// TIA Portal project "FactoryIO_Template_S7-1200_V16_V16" (V16)
// Vorlageprojekt für das Buch mit Zielsystem S7-1200

(* hardware
DEVICE "S7-1200-Station_1"  S7-1200 Station
   slot 0: "Baugruppenträger_0"  Rack  V1.0
   slot 1: "PLC_1"  CPU 1211C DC/DC/DC  6ES7 211-1AE40-0XB0  V4.1
*)

// ===== PLC "PLC_1"  CPU 1211C DC/DC/DC =====

VAR_GLOBAL   // PLC tag table "Standard-Variablentabelle"
   "Start" AT %I0.0 : Bool;
   "stop" AT %I0.1 : Bool;
   "Vsion_top" AT %I0.2 : Bool;
   "Vision_base" AT %I0.3 : Bool;
   "Pusher_front_L_base" AT %I0.4 : Bool;
   "Pusher_back_L_base" AT %I0.5 : Bool;
   "Pusher_front_L_top" AT %I0.6 : Bool;
   "Pusher_back_L_top" AT %I0.7 : Bool;
   "Diff_base_pusher" AT %I1.0 : Bool;
   "Diff_top_pusher" AT %I1.1 : Bool;
   "clamped_base" AT %I1.2 : Bool;
   "clamped_top" AT %I1.3 : Bool;
   "Diff_Item_arm" AT %I1.4 : Bool;
   "Move_Z_sensor" AT %I1.5 : Bool;
   "Move_X_sensor" AT %I1.6 : Bool;
   "Diff_base_clamp" AT %I1.7 : Bool;
   "Diff_top_clamp" AT %I2.0 : Bool;
   "Diff_item_leave" AT %I2.1 : Bool;
   "belte_main" AT %Q0.0 : Bool;
   "belte_pushers" AT %Q0.1 : Bool;
   "pusher_base" AT %Q0.2 : Bool;
   "Pusher_top" AT %Q0.3 : Bool;
   "Belte_base" AT %Q0.4 : Bool;
   "Belte_top" AT %Q0.5 : Bool;
   "clamp_base" AT %Q0.6 : Bool;
   "clamp_top" AT %Q0.7 : Bool;
   "up_base" AT %Q1.0 : Bool;
   "Move_z" AT %Q1.1 : Bool;
   "Move_x" AT %Q1.2 : Bool;
   "Grap" AT %Q1.3 : Bool;
   "X" AT %M0.0 : Bool;
   "base" AT %M0.1 : Bool;
   "top" AT %M0.2 : Bool;
   "leave" AT %M0.3 : Bool;
END_VAR

// folder: System blocks/Program resources

DATA_BLOCK "hold_base"   // DB1
{ S7_Optimized_Access := 'TRUE' }
AUTHOR : Simatic
FAMILY : IEC
NAME : IEC_TMR
VERSION : 1.0
// stored: InstanceOfName IEC_TIMER
"IEC_TIMER"
BEGIN
END_DATA_BLOCK

DATA_BLOCK "hold_top"   // DB2
{ S7_Optimized_Access := 'TRUE' }
AUTHOR : Simatic
FAMILY : IEC
NAME : IEC_TMR
VERSION : 1.0
// stored: InstanceOfName IEC_TIMER
"IEC_TIMER"
BEGIN
END_DATA_BLOCK

DATA_BLOCK "wait_for Grap"   // DB3
{ S7_Optimized_Access := 'TRUE' }
AUTHOR : Simatic
FAMILY : IEC
NAME : IEC_TMR
VERSION : 1.0
// stored: InstanceOfName IEC_TIMER
"IEC_TIMER"
BEGIN
END_DATA_BLOCK

DATA_BLOCK "hold_down"   // DB4
{ S7_Optimized_Access := 'TRUE' }
AUTHOR : Simatic
FAMILY : IEC
NAME : IEC_TMR
VERSION : 1.0
// stored: InstanceOfName IEC_TIMER
"IEC_TIMER"
BEGIN
END_DATA_BLOCK

DATA_BLOCK "hold_clamp"   // DB5
{ S7_Optimized_Access := 'TRUE' }
AUTHOR : Simatic
FAMILY : IEC
NAME : IEC_TMR
VERSION : 1.0
// stored: InstanceOfName IEC_TIMER
"IEC_TIMER"
BEGIN
END_DATA_BLOCK

DATA_BLOCK "hlod_base"   // DB6
{ S7_Optimized_Access := 'TRUE' }
AUTHOR : Simatic
FAMILY : IEC
NAME : IEC_TMR
VERSION : 1.0
// stored: InstanceOfName IEC_TIMER
"IEC_TIMER"
BEGIN
END_DATA_BLOCK

DATA_BLOCK "up_hold"   // DB7
{ S7_Optimized_Access := 'TRUE' }
AUTHOR : Simatic
FAMILY : IEC
NAME : IEC_TMR
VERSION : 1.0
// stored: InstanceOfName IEC_TIMER
"IEC_TIMER"
BEGIN
END_DATA_BLOCK

DATA_BLOCK "hold_leave"   // DB8
{ S7_Optimized_Access := 'TRUE' }
AUTHOR : Simatic
FAMILY : IEC
NAME : IEC_TMR
VERSION : 1.0
// stored: InstanceOfName IEC_TIMER
"IEC_TIMER"
BEGIN
END_DATA_BLOCK

// folder: (top level)

FUNCTION "MHJ-PLC-Lab-Function-S71200" : Void   // FC9000, SCL
{ S7_Optimized_Access := 'TRUE' }
VERSION : 0.1
   VAR_TEMP
      rdTimeReturn : Int;
      outputTime : DTL;
      SyncVal : Byte;
      forVal : Int;
      forVal_2 : Int;
      Value : Byte;
   END_VAR
   VAR CONSTANT
      CompVal : Byte := 16#34;
      Value_01 : Byte := 16#11;
      Value_01_DW : DWord := 16#A165_D992;
      Value_02_DW : DWord := 16#58BE_4401;
   END_VAR
BEGIN

   #Value:=PEEK(area := 16#82,
        dbNumber := 0,
        byteOffset := 511);
   #Value := #Value + 1;

   POKE(area := 16#82,
        dbNumber := 0,
        byteOffset := 511,
        value := #Value);

   POKE(area:=16#81,
        dbNumber:=0,
        byteOffset:=1016,
        value:=#Value_01_DW);
   POKE(area := 16#81,
        dbNumber := 0,
        byteOffset := 1020,
        value := #Value_02_DW);

   POKE(area := 16#81,
        dbNumber := 0,
        byteOffset := 511,
        value := B#16#00);

   FOR #forVal := 0 TO 120 DO
       FOR #forVal_2:=0 TO 10 DO
           #rdTimeReturn:=RD_SYS_T(#outputTime);
           #rdTimeReturn := WR_SYS_T(#outputTime);
           #rdTimeReturn := RD_SYS_T(#outputTime);
           #rdTimeReturn := WR_SYS_T(#outputTime);
       END_FOR;
       #SyncVal:= PEEK(area := 16#81,
                      dbNumber := 0,
                      byteOffset := 511);
       IF #SyncVal = #CompVal THEN
          GOTO M_1;
       END_IF;
   END_FOR;
   RETURN;

   M_1:
   POKE(area := 16#81,
        dbNumber := 0,
        byteOffset := 511,
        value := B#16#0);
END_FUNCTION

ORGANIZATION_BLOCK "Main"   // OB1, LAD, ProgramCycle
TITLE = "Main Program Sweep (Cycle)"
{ S7_Optimized_Access := 'TRUE' }
VERSION : 0.1
   VAR_INPUT
      Initial_Call : Bool;   // Initial call of this OB
      Remanence : Bool;   // =True, if remanent data are available
   END_VAR
   VAR_TEMP   // added for the SCL form of the ladder/FBD networks
      _w1 : Bool;
   END_VAR
BEGIN

REGION Network 1: Konnektierungsbaustein für PLC-Lab
   // Im Netzwerk 1 wird der Konnektierungsbaustein für PLC-Lab aufgerufen.
   // Dieser Aufruf darf nicht entfernt werden!
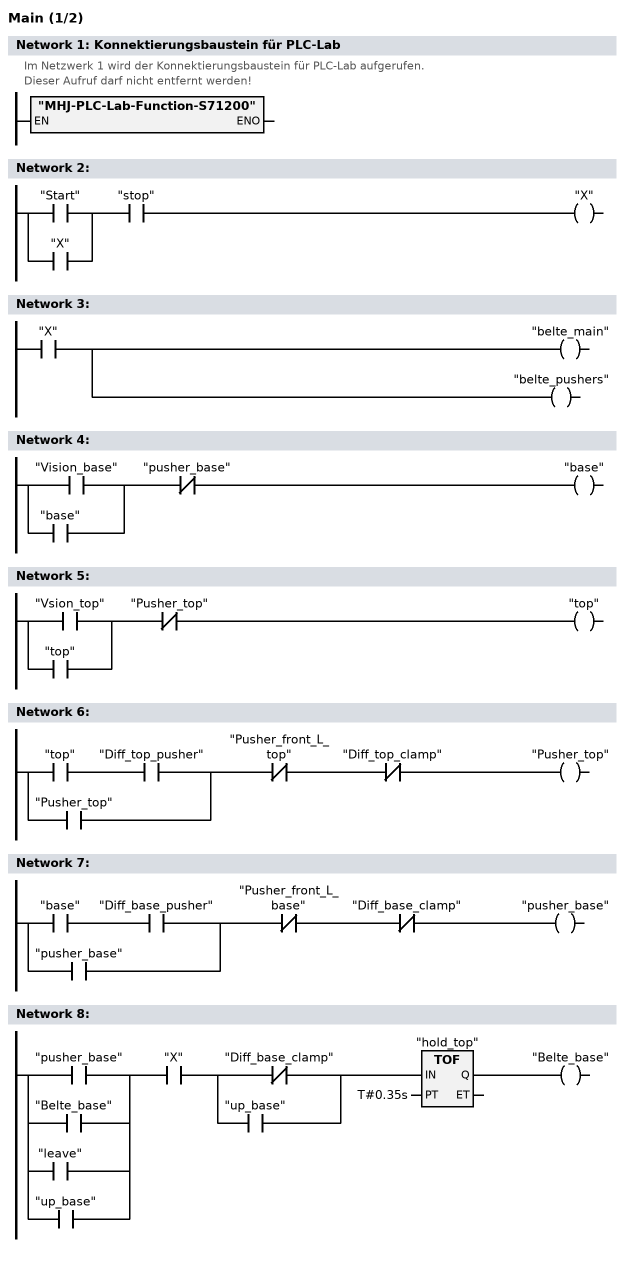
   RUNG wire#powerrail
      "MHJ-PLC-Lab-Function-S71200"()
   END_RUNG
   // the same network as SCL:
   "MHJ-PLC-Lab-Function-S71200"();
END_REGION

REGION Network 2
   RUNG wire#powerrail
      Contact( "Start" )
      wire#w1
      Contact( "stop" )
      Coil( "X" )
   END_RUNG
   RUNG wire#powerrail
      Contact( "X" )
   END_RUNG wire#w1
   // the same network as SCL:
   "X" := ("Start" OR "X") AND "stop";
END_REGION

REGION Network 3
   RUNG wire#powerrail
      Contact( "X" )
      wire#w1
      Coil( "belte_main" )
   END_RUNG
   RUNG wire#w1
      Coil( "belte_pushers" )
   END_RUNG
   // the same network as SCL:
   "belte_main" := "X";
   "belte_pushers" := "X";
END_REGION

REGION Network 4
   RUNG wire#powerrail
      Contact( "Vision_base" )
      wire#w1
      I_Contact( "pusher_base" )
      Coil( "base" )
   END_RUNG
   RUNG wire#powerrail
      Contact( "base" )
   END_RUNG wire#w1
   // the same network as SCL:
   "base" := ("Vision_base" OR "base") AND NOT "pusher_base";
END_REGION

REGION Network 5
   RUNG wire#powerrail
      Contact( "Vsion_top" )
      wire#w1
      I_Contact( "Pusher_top" )
      Coil( "top" )
   END_RUNG
   RUNG wire#powerrail
      Contact( "top" )
   END_RUNG wire#w1
   // the same network as SCL:
   "top" := ("Vsion_top" OR "top") AND NOT "Pusher_top";
END_REGION

REGION Network 6
   RUNG wire#powerrail
      Contact( "top" )
      Contact( "Diff_top_pusher" )
      wire#w1
      I_Contact( "Pusher_front_L_top" )
      I_Contact( "Diff_top_clamp" )
      Coil( "Pusher_top" )
   END_RUNG
   RUNG wire#powerrail
      Contact( "Pusher_top" )
   END_RUNG wire#w1
   // the same network as SCL:
   "Pusher_top" := (("top" AND "Diff_top_pusher") OR "Pusher_top") AND NOT "Pusher_front_L_top" AND NOT "Diff_top_clamp";
END_REGION

REGION Network 7
   RUNG wire#powerrail
      Contact( "base" )
      Contact( "Diff_base_pusher" )
      wire#w1
      I_Contact( "Pusher_front_L_base" )
      I_Contact( "Diff_base_clamp" )
      Coil( "pusher_base" )
   END_RUNG
   RUNG wire#powerrail
      Contact( "pusher_base" )
   END_RUNG wire#w1
   // the same network as SCL:
   "pusher_base" := (("base" AND "Diff_base_pusher") OR "pusher_base") AND NOT "Pusher_front_L_base" AND NOT "Diff_base_clamp";
END_REGION

REGION Network 8
   "hold_top".TOF(IN := ("pusher_base" OR "Belte_base" OR "leave" OR "up_base") AND "X" AND (NOT "Diff_base_clamp" OR "up_base"),
                  PT := T#0.35s);
   "Belte_base" := "hold_top".Q;
END_REGION

REGION Network 9
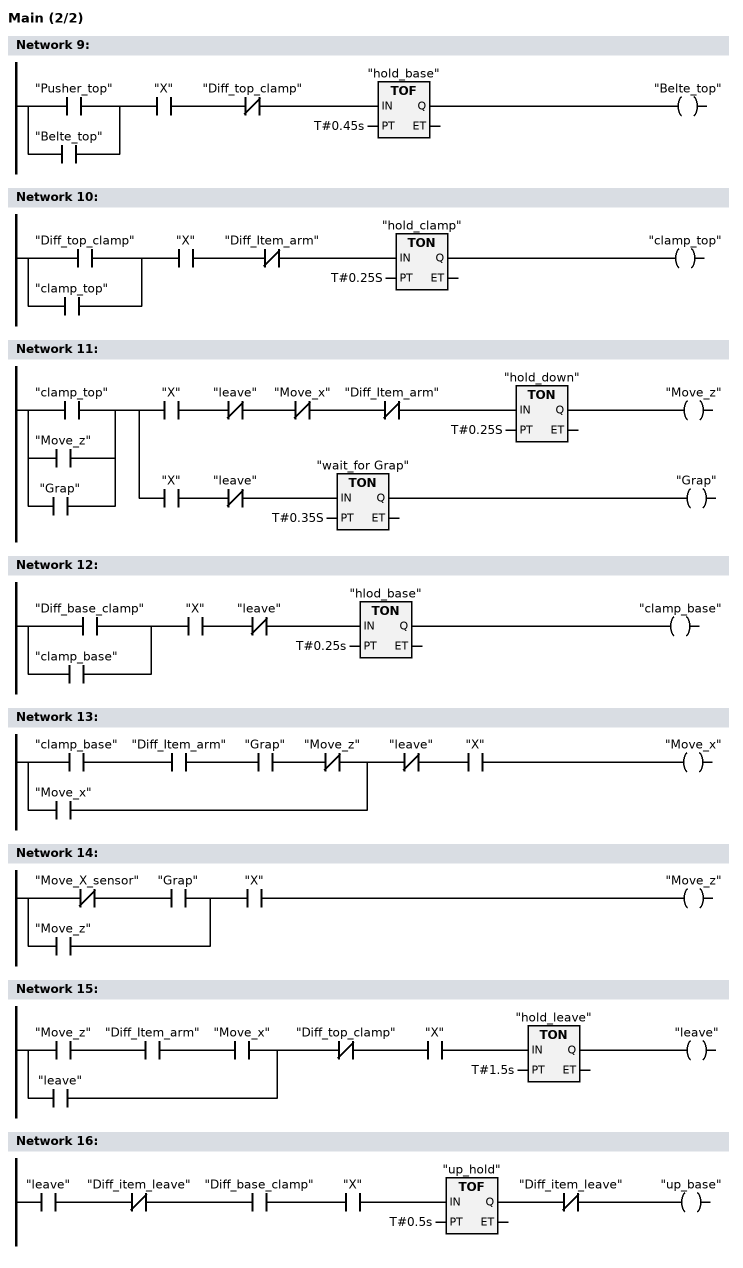
   "hold_base".TOF(IN := ("Pusher_top" OR "Belte_top") AND "X" AND NOT "Diff_top_clamp", PT := T#0.45s);
   "Belte_top" := "hold_base".Q;
END_REGION

REGION Network 10
   "hold_clamp".TON(IN := ("Diff_top_clamp" OR "clamp_top") AND "X" AND NOT "Diff_Item_arm", PT := T#0.25S);
   "clamp_top" := "hold_clamp".Q;
END_REGION

REGION Network 11
   #_w1 := "clamp_top" OR "Move_z" OR "Grap";
   "hold_down".TON(IN := #_w1 AND "X" AND NOT "leave" AND NOT "Move_x" AND NOT "Diff_Item_arm", PT := T#0.25S);
   "Move_z" := "hold_down".Q;
   "wait_for Grap".TON(IN := #_w1 AND "X" AND NOT "leave", PT := T#0.35S);
   "Grap" := "wait_for Grap".Q;
END_REGION

REGION Network 12
   "hlod_base".TON(IN := ("Diff_base_clamp" OR "clamp_base") AND "X" AND NOT "leave", PT := T#0.25s);
   "clamp_base" := "hlod_base".Q;
END_REGION

REGION Network 13
   RUNG wire#powerrail
      Contact( "clamp_base" )
      Contact( "Diff_Item_arm" )
      Contact( "Grap" )
      I_Contact( "Move_z" )
      wire#w1
      I_Contact( "leave" )
      Contact( "X" )
      Coil( "Move_x" )
   END_RUNG
   RUNG wire#powerrail
      Contact( "Move_x" )
   END_RUNG wire#w1
   // the same network as SCL:
   "Move_x" := (("clamp_base" AND "Diff_Item_arm" AND "Grap" AND NOT "Move_z") OR "Move_x") AND NOT "leave" AND "X";
END_REGION

REGION Network 14
   RUNG wire#powerrail
      I_Contact( "Move_X_sensor" )
      Contact( "Grap" )
      wire#w1
      Contact( "X" )
      Coil( "Move_z" )
   END_RUNG
   RUNG wire#powerrail
      Contact( "Move_z" )
   END_RUNG wire#w1
   // the same network as SCL:
   "Move_z" := ((NOT "Move_X_sensor" AND "Grap") OR "Move_z") AND "X";
END_REGION

REGION Network 15
   "hold_leave".TON(IN := (("Move_z" AND "Diff_Item_arm" AND "Move_x") OR "leave") AND NOT "Diff_top_clamp" AND "X",
                    PT := T#1.5s);
   "leave" := "hold_leave".Q;
END_REGION

REGION Network 16
   "up_hold".TOF(IN := "leave" AND NOT "Diff_item_leave" AND "Diff_base_clamp" AND "X", PT := T#0.5s);
   "up_base" := "up_hold".Q AND NOT "Diff_item_leave";
END_REGION
END_ORGANIZATION_BLOCK